TYPE Auto_Test_DUT :
STRUCT
	Duration:	TIME;
	Start_Time:	STRING[20];
	Stop_Time:	STRING[20];
	Time_Running:	TIME;
	Total_Duration:	TIME;
END_STRUCT
END_TYPE

(* stored: Version 1.1.0.1
   DUT Auto_Test_DUT: Id {cc0272a1-c3cc-4742-8c49-9f64db54f5c6} *)
